Universal Robots PolyScope program: SUB_7001.urp

Program SUB_7001 (installation=GD directory=/programs/GD createdIn=5.13.0 lastSavedIn=5.13.0 robotSerialNumber=20205000017)
Calibrated DH parameters: a=[-0.000157, -0.56303, -0.236706, -0.000074, -0.000109, 0]; d=[0.181705, 47.632387, 369.599619, -417.058513, 0.119878, 0.115667]; alpha=[1.570881, -0.005074, -0.001247, 1.56886, -1.570997, 0]; deltaTheta=[0, -0.405485, 5.544791, 1.143886, -0.000009, -0.000001]
InitVariablesNode
Robot Program (runOnlyOnce=false)
  SetPayload (workpieceName=k10)
  MoveL speed 120 mm/s, acceleration 70 mm/s^2 (useActiveTCP=false) tcp=TCP_1; feature=Base
    Waypoint Variable (Variable): variable(featureName=gTAIHI_pos1)
    Waypoint Variable (Variable): variable(featureName=gTAIHI_pos2)
    Waypoint Variable (Variable): variable(featureName=gTAIHI_pos3)
    Waypoint Variable (Variable): variable(featureName=gTAIHI_pos4)
    SetPayload (workpieceName=k120)
    Waypoint Variable (Variable): variable(featureName=gTAIHI_pos5)
    Folder FREE_DRIVE
      SetPayload (workpieceName=k2)
      Script: freedrive_mode()
      Set NoAction tcp=ZERO
      Wait Sleep waitTime=0.5
      Script: end_freedrive_mode()
